# EPICS substitutions: ek9000App/Db/EL3311.substitutions
file EL3311.template
{       pattern
        {
                TERMINAL,

        }
        {
        }
}
